PROGRAM MAIN_TCP
VAR
	//TCP/IP Comunicacion
	s_IP			: STRING(15) := '192.168.1.138';
	udi_Port		: UDINT := 2000;
	fbServer 		: Fagor_ServidorLocalTCP;
	bEnableServer	: BOOL;
	
	fbSocketCloseAll: FB_SocketCloseAll;
	bCloseAll 		: BOOL;

	bResetGeneral: BOOL;
END_VAR

// CONTROL DEL SERVIDOR
bEnableServer 		:= bEnableServer;		//Habilitar servidor
s_IP 				:= s_IP;				//IP local de la máquina (en caso de ser servidor).
udi_Port			:= udi_Port;			//Puerto local de la máquina (en caso de ser servidor)
G_bLogDebugMessages := G_bLogDebugMessages;	//Mostrar mensajes de debug en la consola
G_bLogErrorMessages	:= G_bLogErrorMessages;	//Mostrar mensajes de error en la consola

// RESET
bResetGeneral := bResetGeneral;

// CERRAR TODAS LAS CONEXIONES
bCloseAll := bCloseAll;

IF bCloseAll THEN 
	fbSocketCloseAll( 
					bExecute	:= TRUE
					,sSrvNetId 	:= ''
					,tTimeout 	:= T#3S 
					);
	IF NOT fbSocketCloseAll.bBusy THEN
		IF NOT fbSocketCloseAll.bError THEN
			bCloseAll := FALSE;
		ELSE
			fbSocketCloseAll(bExecute := TRUE );			
		END_IF
	END_IF
END_IF
fbSocketCloseAll( bExecute:= FALSE );

IF NOT fbSocketCloseAll.bBusy THEN
	fbServer( 	bEnable 	:= bEnableServer
				,sLocalHost := s_IP
				,nLocalPort := udi_Port
				,bReset 	:= bResetGeneral );
END_IF
bResetGeneral := FALSE;

END_PROGRAM

(* stored: Version 1.1.0.1, ProductVersion 3.1.4024.3
   POU MAIN_TCP: Id {f90a88f7-c38f-4499-8154-44cceb8647d5}, SpecialFunc None *)
